   REGION "MB3 Code 4071-  MANIPOLATORE -AX"
      A03_HMI.MB3.Button.A0302.Manipolatore.Ax.Bwd_Minus := ((MB3_Decoder.Code = #4071_MANIPOLATORE_AX) AND MB3_Decoder.OperationMinus);
      A03_HMI.MB3.Button.A0302.Manipolatore.Ax.Fwd_Plus := ((MB3_Decoder.Code = #4071_MANIPOLATORE_AX) AND MB3_Decoder.OperationPlus);
      IF (((((MB3_Decoder.Code = #4071_MANIPOLATORE_AX) AND A0302_Manipolatore.COut.Testa.Ax.MinusCheckNext) OR ((MB3_Decoder.Code = #4071_MANIPOLATORE_AX) AND A0302_Manipolatore.COut.Coda.Ax.MinusCheckNext)) AND A03_HMI.MB3.Button.A0302.Manipolatore.Ax.Bwd_Minus) OR ((((MB3_Decoder.Code = #4071_MANIPOLATORE_AX) AND A0302_Manipolatore.COut.Testa.Ax.PlusCheckNext) OR ((MB3_Decoder.Code = #4071_MANIPOLATORE_AX) AND A0302_Manipolatore.COut.Coda.Ax.PlusCheckNext)) AND A03_HMI.MB3.Button.A0302.Manipolatore.Ax.Fwd_Plus)) THEN
         MB3_Decoder.OpEnabled := TRUE;
      END_IF;
      IF (((MB3_Decoder.Code = #4071_MANIPOLATORE_AX) AND NOT (A0302_Manipolatore.COut.Testa.Ax.Standstill)) OR ((MB3_Decoder.Code = #4071_MANIPOLATORE_AX) AND NOT (A0302_Manipolatore.COut.Coda.Ax.Standstill))) THEN
         MB3_Decoder.OpRunning := TRUE;
      END_IF;
      IF ((MB3_Decoder.Code = #4071_MANIPOLATORE_AX) AND FALSE) THEN
         MB3_Decoder.OpDone := TRUE;
      END_IF;
   END_REGION

   REGION "MB3 Code 4072-  MANIPOLATORE -AX-POS"
      A03_HMI.MB3.Button.A0302.Manipolatore.Ax.MoveToPos := ((((MB3_Decoder.Code = #4072_MANIPOLATORE_AX-POS) AND (A0302_Manipolatore.Ax_Testa.COut.ActualPosition <> A0302_Manipolatore.Ax_Testa.HMI.Sts.TargetPos)) OR ((MB3_Decoder.Code = #4072_MANIPOLATORE_AX-POS) AND (A0302_Manipolatore.Ax_Coda.COut.ActualPosition <> A0302_Manipolatore.Ax_Coda.HMI.Sts.TargetPos))) AND MB3_Decoder.OperationPlus);
      IF ((((MB3_Decoder.Code = #4072_MANIPOLATORE_AX-POS) AND A0302_Manipolatore.COut.Testa.Ax.MinusCheckNext) OR ((MB3_Decoder.Code = #4072_MANIPOLATORE_AX-POS) AND A0302_Manipolatore.COut.Coda.Ax.MinusCheckNext) OR ((MB3_Decoder.Code = #4072_MANIPOLATORE_AX-POS) AND A0302_Manipolatore.COut.Testa.Ax.PlusCheckNext) OR ((MB3_Decoder.Code = #4072_MANIPOLATORE_AX-POS) AND A0302_Manipolatore.COut.Coda.Ax.PlusCheckNext)) AND A03_HMI.MB3.Button.A0302.Manipolatore.Ax.MoveToPos) THEN
         MB3_Decoder.OpEnabled := TRUE;
      END_IF;
      IF (((MB3_Decoder.Code = #4072_MANIPOLATORE_AX-POS) AND NOT (A0302_Manipolatore.COut.Testa.Ax.Standstill)) OR ((MB3_Decoder.Code = #4072_MANIPOLATORE_AX-POS) AND NOT (A0302_Manipolatore.COut.Coda.Ax.Standstill))) THEN
         MB3_Decoder.OpRunning := TRUE;
      END_IF;
      IF (((MB3_Decoder.Code = #4072_MANIPOLATORE_AX-POS) AND A0302_Manipolatore.Ax_Testa.COut.InPosition) AND A0302_Manipolatore.Ax_Coda.COut.InPosition) THEN
         MB3_Decoder.OpDone := TRUE;
      END_IF;
   END_REGION

   REGION "MB3 Code 4073 - MANIPOLATORE- MAGNETE"
      A03_HMI.MB3.Button.A0302.Manipolatore.Magnete.Rest := ((MB3_Decoder.Code = #4073_MANIPOLATORE_MAGNETE) AND MB3_Decoder.OperationMinus);
      A03_HMI.MB3.Button.A0302.Manipolatore.Magnete.Work := ((MB3_Decoder.Code = #4073_MANIPOLATORE_MAGNETE) AND MB3_Decoder.OperationPlus);
      IF (((((MB3_Decoder.Code = #4073_MANIPOLATORE_MAGNETE) AND A0302_Manipolatore.COut.Testa.Magnete.Rest_CheckNext) OR ((MB3_Decoder.Code = #4073_MANIPOLATORE_MAGNETE) AND A0302_Manipolatore.COut.Coda.Magnete.Rest_CheckNext)) AND A03_HMI.MB3.Button.A0302.Manipolatore.Magnete.Rest) OR ((((MB3_Decoder.Code = #4073_MANIPOLATORE_MAGNETE) AND A0302_Manipolatore.COut.Testa.Magnete.Work_CheckNext) OR ((MB3_Decoder.Code = #4073_MANIPOLATORE_MAGNETE) AND A0302_Manipolatore.COut.Testa.Magnete.Rest_CheckNext)) AND A03_HMI.MB3.Button.A0302.Manipolatore.Magnete.Work)) THEN
         MB3_Decoder.OpEnabled := TRUE;
      END_IF;
      IF (((MB3_Decoder.Code = #4073_MANIPOLATORE_MAGNETE) AND NOT (A0302_Manipolatore.COut.Testa.Magnete.Standstill)) OR ((MB3_Decoder.Code = #4073_MANIPOLATORE_MAGNETE) AND NOT (A0302_Manipolatore.COut.Coda.Magnete.Standstill))) THEN
         MB3_Decoder.OpRunning := TRUE;
      END_IF;
      IF ((((MB3_Decoder.Code = #4073_MANIPOLATORE_MAGNETE) AND A03_HMI.MB3.Button.A0302.Manipolatore.Magnete.Rest) AND A0302_Manipolatore.COut.Testa.Magnete.Rest) OR (((MB3_Decoder.Code = #4073_MANIPOLATORE_MAGNETE) AND A03_HMI.MB3.Button.A0302.Manipolatore.Magnete.Rest) AND A0302_Manipolatore.COut.Coda.Magnete.Rest) OR (((MB3_Decoder.Code = #4073_MANIPOLATORE_MAGNETE) AND A03_HMI.MB3.Button.A0302.Manipolatore.Magnete.Work) AND A0302_Manipolatore.COut.Testa.Magnete.Work) OR (((MB3_Decoder.Code = #4073_MANIPOLATORE_MAGNETE) AND A03_HMI.MB3.Button.A0302.Manipolatore.Magnete.Work) AND A0302_Manipolatore.COut.Coda.Magnete.Work)) THEN
         MB3_Decoder.OpDone := TRUE;
      END_IF;
   END_REGION

   REGION "MB3 Code 4074 - MANIPOLATORE- SOLLEVATORE"
      A03_HMI.MB3.Button.A0302.Manipolatore.Sollevatore.Rest := ((MB3_Decoder.Code = #4074_MANIPOLATORE_SOLLEVATORE) AND MB3_Decoder.OperationMinus);
      A03_HMI.MB3.Button.A0302.Manipolatore.Sollevatore.Work := ((MB3_Decoder.Code = #4074_MANIPOLATORE_SOLLEVATORE) AND MB3_Decoder.OperationPlus);
      IF (((((MB3_Decoder.Code = #4074_MANIPOLATORE_SOLLEVATORE) AND A0302_Manipolatore.COut.Testa.Sollevatore.Rest_CheckNext) OR ((MB3_Decoder.Code = #4074_MANIPOLATORE_SOLLEVATORE) AND A0302_Manipolatore.COut.Coda.Sollevatore.Rest_CheckNext)) AND A03_HMI.MB3.Button.A0302.Manipolatore.Sollevatore.Rest) OR ((((MB3_Decoder.Code = #4074_MANIPOLATORE_SOLLEVATORE) AND A0302_Manipolatore.COut.Testa.Sollevatore.Work_CheckNext) OR ((MB3_Decoder.Code = #4074_MANIPOLATORE_SOLLEVATORE) AND A0302_Manipolatore.COut.Testa.Sollevatore.Rest_CheckNext)) AND A03_HMI.MB3.Button.A0302.Manipolatore.Sollevatore.Work)) THEN
         MB3_Decoder.OpEnabled := TRUE;
      END_IF;
      IF (((MB3_Decoder.Code = #4074_MANIPOLATORE_SOLLEVATORE) AND NOT (A0302_Manipolatore.COut.Testa.Sollevatore.Standstill)) OR ((MB3_Decoder.Code = #4074_MANIPOLATORE_SOLLEVATORE) AND NOT (A0302_Manipolatore.COut.Coda.Sollevatore.Standstill))) THEN
         MB3_Decoder.OpRunning := TRUE;
      END_IF;
      IF ((((MB3_Decoder.Code = #4074_MANIPOLATORE_SOLLEVATORE) AND A03_HMI.MB3.Button.A0302.Manipolatore.Sollevatore.Rest) AND A0302_Manipolatore.COut.Testa.Sollevatore.Rest) OR (((MB3_Decoder.Code = #4074_MANIPOLATORE_SOLLEVATORE) AND A03_HMI.MB3.Button.A0302.Manipolatore.Sollevatore.Rest) AND A0302_Manipolatore.COut.Coda.Sollevatore.Rest) OR (((MB3_Decoder.Code = #4074_MANIPOLATORE_SOLLEVATORE) AND A03_HMI.MB3.Button.A0302.Manipolatore.Sollevatore.Work) AND A0302_Manipolatore.COut.Testa.Sollevatore.Work) OR (((MB3_Decoder.Code = #4074_MANIPOLATORE_SOLLEVATORE) AND A03_HMI.MB3.Button.A0302.Manipolatore.Sollevatore.Work) AND A0302_Manipolatore.COut.Coda.Sollevatore.Work)) THEN
         MB3_Decoder.OpDone := TRUE;
      END_IF;
   END_REGION

   REGION "MB3 Decoder"
      #MB3_Decoder(
         en := TRUE,
         ButtonMinus := NOT ((NOT (MB3_Pb_Comando_Manuale_Jog_Minus_A03) AND NOT (A03_HMI.Area03.SuperUser.JogMinus))),
         ButtonPlus := NOT ((NOT (MB3_Pb_Comando_Manuale_Jog_Plus_A03) AND NOT (A03_HMI.Area03.SuperUser.JogPlus))),
         CodeReq := A03_HMI.MB3.ManCode_REQ,
         Code => A03_HMI.MB3.ManCode_CMD,
         Lamp => MB3_LpJog
      );

      #MB3_Decoder.Q;
   END_REGION


END_FUNCTION_BLOCK
